{attribute 'GeneratedUsingTerminal: EK1100-0000-0018'}
{attribute addProperty BoxType "EK1100-0000-0018"}
{attribute addProperty Id "Beckhoff_EJ3xxxEK1122Beckhoff_EJ3xxxEK1122_1A5DA9A52A_0001_EJ3004_0000_0019EJ3004_C4269E3248A_0002_EJ3004_0000_0020EJ3004_C4269E3248A_0003_EJ3004_0000_0021EJ3004_C4269E3248A_0004_EJ3048_0000_0020EJ3048_335F857B84A_0005_EJ3058_0000_0020EJ3058_335F857B84A_0006_EJ3068_0000_0020EJ3068_335F857B84A_0007_EJ3068_0000_0021EJ3068_335F857B84A_0008_EJ3104_0000_0019EJ3104_DCC7866252A_0009_EJ3104_0000_0020EJ3104_DCC7866252A_0010_EJ3104_0000_0021EJ3104_DCC7866252A_0011_EJ3108_0000_0017EJ3108_335F857B84A_0012_EJ3108_0000_0018EJ3108_35AE532492A_0013_EJ3108_0000_0019EJ3108_35AE532492A_0014_EJ3202_0000_0019EJ3202_28AA99ED30A_0015_EJ3202_0000_0020EJ3202_28AA99ED30A_0016_EJ3202_0000_0021EJ3202_28AA99ED30A_0017_EJ3214_0000_0016EJ3214_8BBE23EA40A_0018_EJ3255_0000_0023EJ3255_1972F7C062A_0019_EJ3318_0000_0017EJ3318_BD104D8882"}
{attribute addProperty CRC "4224222290"}
{attribute addProperty Size "1180"}
TYPE Beckhoff_EJ3xxx_FBC88452 EXTENDS EK1100_1FC0878B :
STRUCT
	{attribute addProperty Name "Beckhoff_EJ3xxxEK1122"}
	Beckhoff_EJ3xxxEK1122 : Beckhoff_EJ3xxxEK1122_1A5DA9A5;
	{attribute addProperty Name "A_0001_EJ3004_0000_0019"}
	A_0001_EJ3004_0000_0019 : EJ3004_C4269E32;
	{attribute addProperty Name "A_0002_EJ3004_0000_0020"}
	A_0002_EJ3004_0000_0020 : EJ3004_C4269E32;
	{attribute addProperty Name "A_0003_EJ3004_0000_0021"}
	A_0003_EJ3004_0000_0021 : EJ3004_C4269E32;
	{attribute addProperty Name "A_0004_EJ3048_0000_0020"}
	A_0004_EJ3048_0000_0020 : EJ3048_335F857B;
	{attribute addProperty Name "A_0005_EJ3058_0000_0020"}
	A_0005_EJ3058_0000_0020 : EJ3058_335F857B;
	{attribute addProperty Name "A_0006_EJ3068_0000_0020"}
	A_0006_EJ3068_0000_0020 : EJ3068_335F857B;
	{attribute addProperty Name "A_0007_EJ3068_0000_0021"}
	A_0007_EJ3068_0000_0021 : EJ3068_335F857B;
	{attribute addProperty Name "A_0008_EJ3104_0000_0019"}
	A_0008_EJ3104_0000_0019 : EJ3104_DCC78662;
	{attribute addProperty Name "A_0009_EJ3104_0000_0020"}
	A_0009_EJ3104_0000_0020 : EJ3104_DCC78662;
	{attribute addProperty Name "A_0010_EJ3104_0000_0021"}
	A_0010_EJ3104_0000_0021 : EJ3104_DCC78662;
	{attribute addProperty Name "A_0011_EJ3108_0000_0017"}
	A_0011_EJ3108_0000_0017 : EJ3108_335F857B;
	{attribute addProperty Name "A_0012_EJ3108_0000_0018"}
	A_0012_EJ3108_0000_0018 : EJ3108_35AE5324;
	{attribute addProperty Name "A_0013_EJ3108_0000_0019"}
	A_0013_EJ3108_0000_0019 : EJ3108_35AE5324;
	{attribute addProperty Name "A_0014_EJ3202_0000_0019"}
	A_0014_EJ3202_0000_0019 : EJ3202_28AA99ED;
	{attribute addProperty Name "A_0015_EJ3202_0000_0020"}
	A_0015_EJ3202_0000_0020 : EJ3202_28AA99ED;
	{attribute addProperty Name "A_0016_EJ3202_0000_0021"}
	A_0016_EJ3202_0000_0021 : EJ3202_28AA99ED;
	{attribute addProperty Name "A_0017_EJ3214_0000_0016"}
	A_0017_EJ3214_0000_0016 : EJ3214_8BBE23EA;
	{attribute addProperty Name "A_0018_EJ3255_0000_0023"}
	A_0018_EJ3255_0000_0023 : EJ3255_1972F7C0;
	{attribute addProperty Name "A_0019_EJ3318_0000_0017"}
	A_0019_EJ3318_0000_0017 : EJ3318_BD104D88;
END_STRUCT
END_TYPE

(* stored: Version 1.2.0.0, ProductVersion 3.1.4024.9
   DUT Beckhoff_EJ3xxx_FBC88452: Id {07c165d9-e502-4b95-9f39-9f4c6c2182cb} *)
